% RSLogix 500 project P7_IVANOVSKI_M.RSS, saved by version 8.30.00.16 %
PROJECT "UNTITLED"    % processor: Bul.1763 MicroLogix 1100 Series B %

PROGRAM FILES
  LAD 2 "MAIN"  5 rungs
  LAD 3 "CALC"  7 rungs
  LAD 4 "CYCLE"  4 rungs

DATA FILES
  O0 OUTPUT  8 elements
  I1 INPUT  8 elements
  S2 STATUS  66 elements
  B3 BINARY  2 elements
  T4 TIMER  2 elements
  C5 COUNTER  2 elements
  R6 CONTROL  1 elements
  N7 INTEGER  15 elements
  F8 FLOAT  9 elements
  PD9 CONCEN.  1 elements  % O2 CONCENTRATION %

LADDER 2 "MAIN"
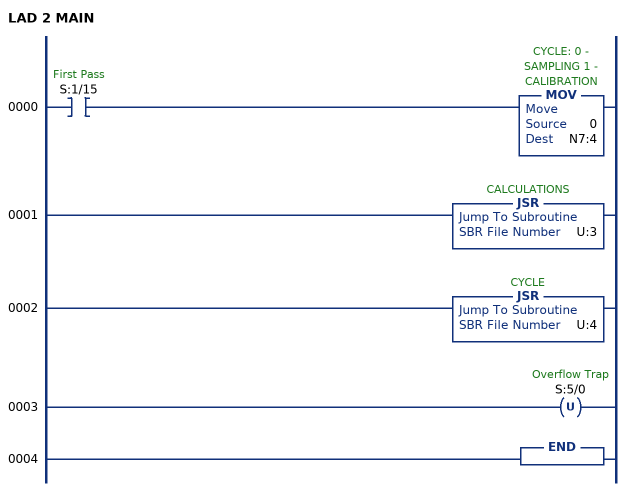
% Rung: 0 %
SOR XIC S:1/15 MOV 0 N7:4 EOR
%   S:1/15  "First Pass" %
%   N7:4  "CYCLE: 0 - SAMPLING 1 - CALIBRATION" %
% Rung: 1 %
SOR JSR U:3 EOR
%   U:3  "CALCULATIONS" %
% Rung: 2 %
SOR JSR U:4 EOR
%   U:4  "CYCLE" %
% Rung: 3 %
SOR OTU S:5/0 EOR
%   S:5/0  "Overflow Trap" %
% Rung: 4 %
SOR END EOR

LADDER 3 "CALC"
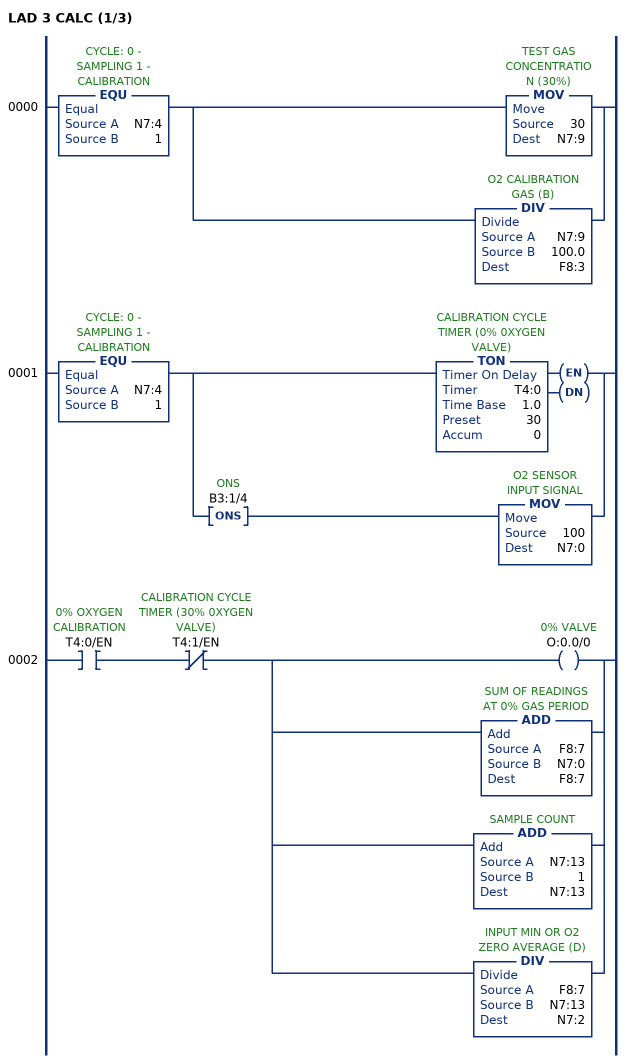
% Rung: 0 %
SOR EQU N7:4 1 BST MOV 30 N7:9 NXB DIV N7:9 100.0 F8:3 BND EOR
%   N7:4  "CYCLE: 0 - SAMPLING 1 - CALIBRATION" %
%   N7:9  "TEST GAS CONCENTRATION (30%)" %
%   F8:3  "O2 CALIBRATION GAS (B)" %
% Rung: 1 %
SOR EQU N7:4 1 BST TON T4:0 1.0 30 0 NXB ONS B3:1/4 MOV 100 N7:0 BND EOR
%   N7:4  "CYCLE: 0 - SAMPLING 1 - CALIBRATION" %
%   T4:0  "CALIBRATION CYCLE TIMER (0% 0XYGEN VALVE)" %
%   B3:1/4  "ONS" %
%   N7:0  "O2 SENSOR INPUT SIGNAL" %
% Rung: 2 %
SOR XIC T4:0/EN XIO T4:1/EN BST OTE O:0.0/0 NXB ADD F8:7 N7:0 F8:7 NXB ADD N7:13 1 N7:13 NXB DIV F8:7 N7:13 N7:2 BND EOR
%   T4:0/EN  "0% OXYGEN CALIBRATION" %
%   T4:1  "CALIBRATION CYCLE TIMER (30% 0XYGEN VALVE)" %
%   O:0.0/0  "0% VALVE" %
%   F8:7  "SUM OF READINGS AT 0% GAS PERIOD" %
%   N7:0  "O2 SENSOR INPUT SIGNAL" %
%   N7:13  "SAMPLE COUNT" %
%   N7:2  "INPUT MIN OR O2 ZERO AVERAGE (D)" %

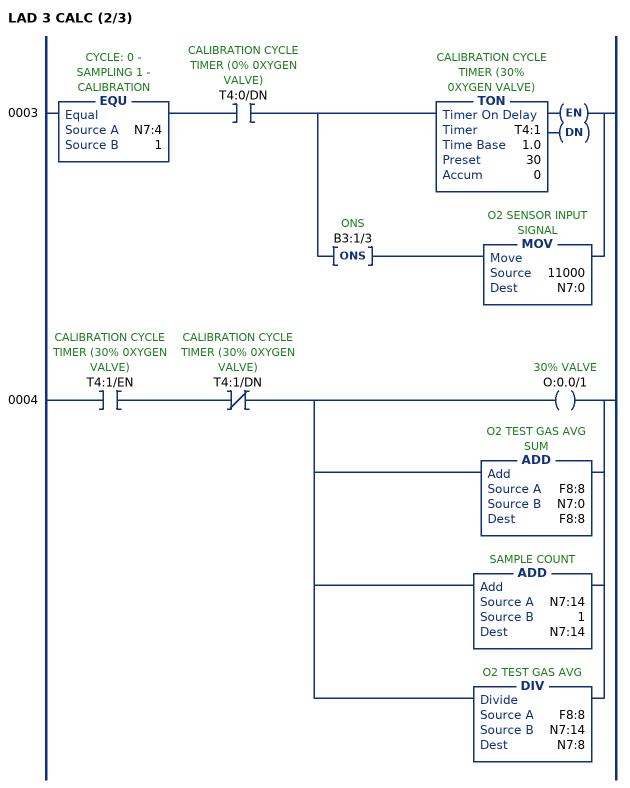
% Rung: 3 %
SOR EQU N7:4 1 XIC T4:0/DN BST TON T4:1 1.0 30 0 NXB ONS B3:1/3 MOV 11000 N7:0 BND EOR
%   N7:4  "CYCLE: 0 - SAMPLING 1 - CALIBRATION" %
%   T4:0  "CALIBRATION CYCLE TIMER (0% 0XYGEN VALVE)" %
%   T4:1  "CALIBRATION CYCLE TIMER (30% 0XYGEN VALVE)" %
%   B3:1/3  "ONS" %
%   N7:0  "O2 SENSOR INPUT SIGNAL" %
% Rung: 4 %
SOR XIC T4:1/EN XIO T4:1/DN BST OTE O:0.0/1 NXB ADD F8:8 N7:0 F8:8 NXB ADD N7:14 1 N7:14 NXB DIV F8:8 N7:14 N7:8 BND EOR
%   T4:1  "CALIBRATION CYCLE TIMER (30% 0XYGEN VALVE)" %
%   O:0.0/1  "30% VALVE" %
%   F8:8  "O2 TEST GAS AVG SUM" %
%   N7:0  "O2 SENSOR INPUT SIGNAL" %
%   N7:14  "SAMPLE COUNT" %
%   N7:8  "O2 TEST GAS AVG" %

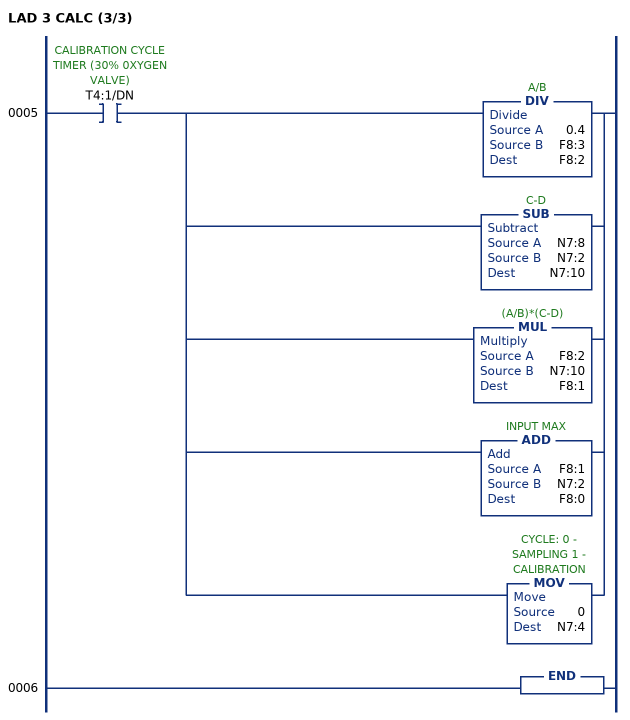
% Rung: 5 %
SOR XIC T4:1/DN BST DIV 0.4 F8:3 F8:2 NXB SUB N7:8 N7:2 N7:10 NXB MUL F8:2 N7:10 F8:1 NXB ADD F8:1 N7:2 F8:0 NXB MOV 0 N7:4 BND EOR
%   T4:1  "CALIBRATION CYCLE TIMER (30% 0XYGEN VALVE)" %
%   F8:3  "O2 CALIBRATION GAS (B)" %
%   F8:2  "A/B" %
%   N7:8  "O2 TEST GAS AVG" %
%   N7:2  "INPUT MIN OR O2 ZERO AVERAGE (D)" %
%   N7:10  "C-D" %
%   F8:1  "(A/B)*(C-D)" %
%   F8:0  "INPUT MAX" %
%   N7:4  "CYCLE: 0 - SAMPLING 1 - CALIBRATION" %
% Rung: 6 %
SOR END EOR

LADDER 4 "CYCLE"
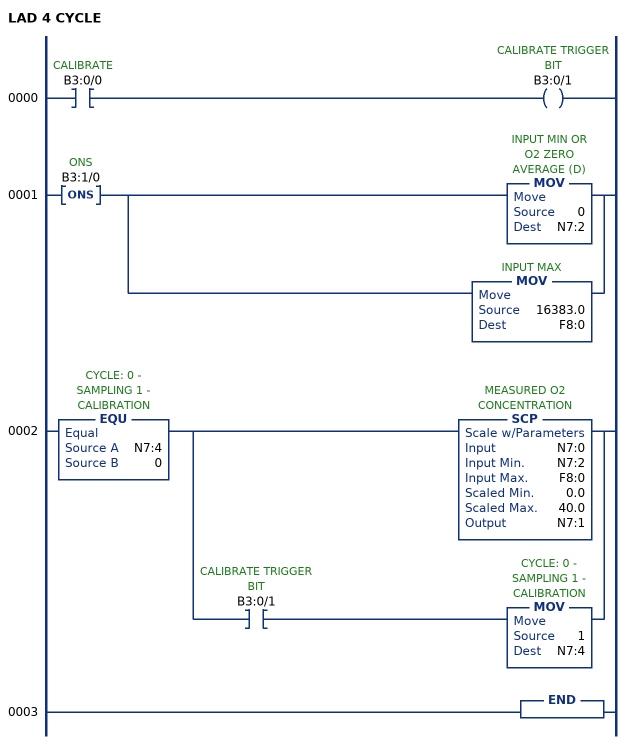
% Rung: 0 %
SOR XIC B3:0/0 OTE B3:0/1 EOR
%   B3:0/0  "CALIBRATE" %
%   B3:0/1  "CALIBRATE TRIGGER BIT" %
% Rung: 1 %
SOR ONS B3:1/0 BST MOV 0 N7:2 NXB MOV 16383.0 F8:0 BND EOR
%   B3:1/0  "ONS" %
%   N7:2  "INPUT MIN OR O2 ZERO AVERAGE (D)" %
%   F8:0  "INPUT MAX" %
% Rung: 2 %
SOR EQU N7:4 0 BST SCP N7:0 N7:2 F8:0 0.0 40.0 N7:1 NXB XIC B3:0/1 MOV 1 N7:4 BND EOR
%   N7:4  "CYCLE: 0 - SAMPLING 1 - CALIBRATION" %
%   N7:0  "O2 SENSOR INPUT SIGNAL" %
%   N7:2  "INPUT MIN OR O2 ZERO AVERAGE (D)" %
%   F8:0  "INPUT MAX" %
%   N7:1  "MEASURED O2 CONCENTRATION" %
%   B3:0/1  "CALIBRATE TRIGGER BIT" %
% Rung: 3 %
SOR END EOR

OTHER DOCUMENTED ADDRESSES
  B3:1/1  "ONS"
  B3:1/2  "ONS"
  B3:1/5  "ONS"
  B3:1/6  "ONS"
  B3:1/7  "ONS"
  C5:0  "ZERO AVG COUNTER"
  C5:0.ACC  "SAMPLING SIZE"
  C5:1  "TEST GAS AVERAGE COUNTER"
  C5:1.ACC  "SAMPLING SIZE"
  F8:4  "O2 MAX CONCENTRATION (A)"
  F8:9  "O2 TEST GAS AVG"
  N7:3  "INPUT MAX (C)"
  N7:5  "O2 MAX CONCENTRATION (40%)"
  N7:7  "02 ZERO AVERAGE"

DATA TABLE (non-zero values as saved)
DATA T4
% .PRE .ACC %
% T4:0 % 30 0
% T4:1 % 30 0
DATA C5
% .PRE .ACC %
% C5:0 % 30 0
% C5:1 % 30 0
